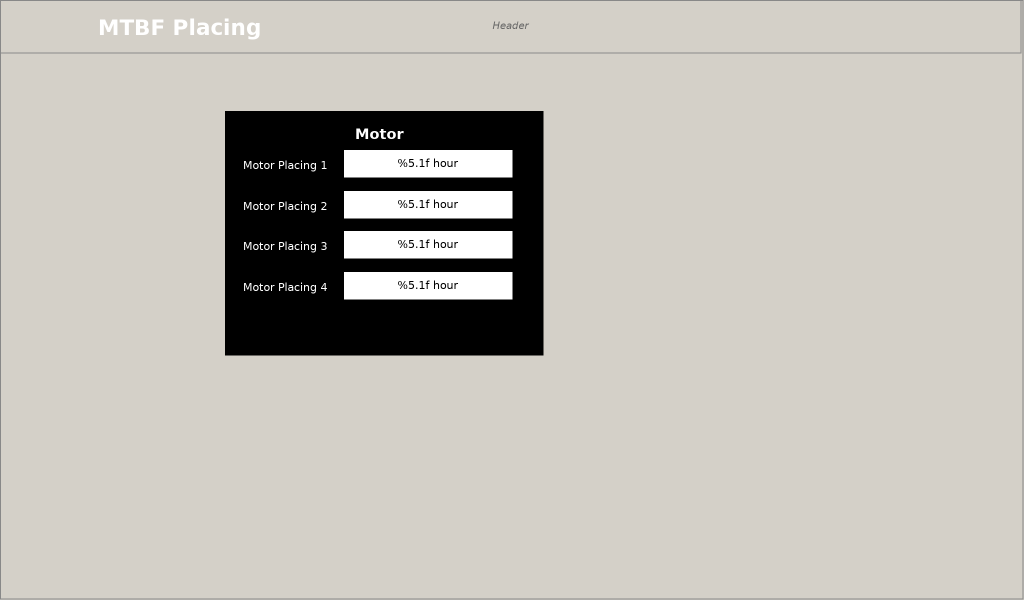
VISUALIZATION MTBF_Placing  // 1024x600
    Frame (0,-2 1021x55)
        shows Header()
    Label (95,15 250x25), "MTBF Placing"
    RoundedRectangle (225,111 318x244)
    Label (243,114 273x40), "Motor"
    Label (240,148 103x35), "Motor Placing 1"
    RoundedRectangle (343,149 170x29), "%5.1f hour", text variable: Status_GVL.stMotor_Placing1.RunningHours
    Label (240,189 103x35), "Motor Placing 2"
    RoundedRectangle (343,190 170x29), "%5.1f hour", text variable: Status_GVL.stMotor_Placing2.RunningHours
    Label (240,229 103x35), "Motor Placing 3"
    RoundedRectangle (343,230 170x29), "%5.1f hour", text variable: Status_GVL.stMotor_Placing3.RunningHours
    Label (240,270 103x35), "Motor Placing 4"
    RoundedRectangle (343,271 170x29), "%5.1f hour", text variable: Status_GVL.stMotor_Placing4.RunningHours
END_VISUALIZATION

(* stored: Version 1.1.0.1, ProductVersion 3.1.4024.12
   Visu MTBF_Placing: Id {06ae5b5e-a293-41a2-8194-5684c7907e5c} *)
